FUNCTION_BLOCK Transition
VAR_INPUT
END_VAR
VAR_OUTPUT
END_VAR
VAR
END_VAR

METHOD WhenGoTo : reference TO Transition
VAR_INPUT
	conditionName	: STRING;
	nextActionName	: STRING;
END_VAR
END_METHOD

END_FUNCTION_BLOCK

(* stored: Version 1.1.0.1, ProductVersion 3.1.4024.11
   POU Transition: Id {ad314cb6-07a4-4fb1-811b-30d8def32fe4}, SpecialFunc None
   Method WhenGoTo: Id {57e063bc-9530-4593-976f-0d6a63848838} *)
